TEXTLIST TextList_Position_Canne
  0 = 'sas' | FR: 'Sas (0)' | EN: 'Loadlock (0)'
  1 = 'egun1' | FR: 'Canon 1' | EN: 'E-gun 1'
  2 = 'evap' | FR: 'Source Joule' | EN: 'Thermal source'
  3 = 'egun2' | FR: 'Canon 2' | EN: 'E-gun 2'
  255 = 'undefined' | FR: 'Indéfinie' | EN: 'Undefined'
   = ''
END_TEXTLIST

(* stored: Version 1.1.0.1, ProductVersion 3.1.4024.10
   TextList TextList_Position_Canne: Id {45116f64-6890-4492-8159-5d37dda89870} *)
